Staubli VAL3: readForce.pgx

program readForce()
begin

  //
  call ati:loopReadForce()

end
